Yaskawa INFORM job: ROBOT2.JBI

/JOB
//NAME ROBOT2
///FOLDERNAME INNE
//POS
///NPOS 25,25,0,0,0,0
///TOOL 0
///POSTYPE PULSE
///PULSE
C00000=-52530,-106772,-59840,25675,74247,58338
C00001=-30541,-61161,-38258,13058,102738,71922
C00002=-79491,-79946,-37138,33739,93735,85492
C00003=-123799,-144126,-48227,54109,53120,88750
C00004=-1049,-85507,-55311,-1240,88725,56676
C00005=10878,-82728,-51898,427,88114,60655
C00006=56233,-75375,-39159,-22430,94952,57482
C00007=77051,-120104,-53646,-32838,65753,47043
C00008=58715,-140663,-55283,-39550,38165,34197
C00009=-10070,-106255,-61443,11351,75991,18903
C00010=4969,-100505,-52101,12303,71167,23538
C00011=24839,-133484,-44655,5407,15605,27035
C00012=51428,-76992,-39319,-14366,84439,67888
C00013=5067,-115869,-54923,15370,51336,49727
C00014=2370,-61149,-31128,13691,95920,53857
C00015=14944,-75662,-39037,14855,81364,56560
C00016=52747,-124419,-44869,-21736,22441,76499
C00017=86721,-65113,-23109,-30643,87847,87051
C00018=67275,-41536,-10599,-20819,100364,86717
C00019=-49708,-95496,-27496,49930,72279,53724
C00020=-14954,-101056,-27545,59819,53704,58945
C00021=-14053,-108943,-20525,82453,42704,47577
C00022=3718,-38650,-2507,33351,95883,82801
C00023=23556,-89945,-42085,25883,63693,43192
C00024=75100,-38847,-12945,-13870,97090,65418
BC00000=140445,1007710,556393
BC00001=140445,1007710,556390
BC00002=140445,1007710,556390
BC00003=140445,1007710,556390
BC00004=140445,1007710,556390
BC00005=140445,1007709,556387
BC00006=140445,1007709,556387
BC00007=140445,1007709,556387
BC00008=140445,1007709,556387
BC00009=140445,1007709,556387
BC00010=140445,1007709,556385
BC00011=140445,1007709,556385
BC00012=140446,1007710,556382
BC00013=140446,1007710,556382
BC00014=140446,1007710,556382
BC00015=140446,1007710,556379
BC00016=140446,1007710,556379
BC00017=140446,1007710,556379
BC00018=140446,1007710,556379
BC00019=140446,1007710,556379
BC00020=140446,1007710,556376
BC00021=140446,1007710,556376
BC00022=140446,1007710,556376
BC00023=140446,1007710,556376
BC00024=140446,1007710,556376
//INST
///DATE 2023/10/04 15:13
///ATTR SC,RW
///GROUP1 RB1,BS1
NOP
*1
MOVJ C00000 BC00000 VJ=0.78 PL=0
MOVJ C00001 BC00001 VJ=0.78 PL=0
MOVJ C00002 BC00002 VJ=0.78 PL=0
MOVJ C00003 BC00003 VJ=0.78 PL=0
MOVJ C00004 BC00004 VJ=0.78 PL=0
*2
MOVJ C00005 BC00005 VJ=0.78 PL=0
MOVJ C00006 BC00006 VJ=0.78 PL=0
MOVJ C00007 BC00007 VJ=0.78 PL=0
MOVJ C00008 BC00008 VJ=0.78 PL=0
MOVJ C00009 BC00009 VJ=0.78 PL=0
*3
MOVJ C00010 BC00010 VJ=0.78 PL=0
MOVJ C00011 BC00011 VJ=0.78 PL=0
MOVJ C00012 BC00012 VJ=0.78 PL=0
MOVJ C00013 BC00013 VJ=0.78 PL=0
MOVJ C00014 BC00014 VJ=0.78 PL=0
*4
MOVJ C00015 BC00015 VJ=0.78 PL=0
MOVJ C00016 BC00016 VJ=0.78 PL=0
MOVJ C00017 BC00017 VJ=0.78 PL=0
MOVJ C00018 BC00018 VJ=0.78 PL=0
MOVJ C00019 BC00019 VJ=0.78 PL=0
*5
MOVJ C00020 BC00020 VJ=0.78 PL=0
MOVJ C00021 BC00021 VJ=0.78 PL=0
MOVJ C00022 BC00022 VJ=0.78 PL=0
MOVJ C00023 BC00023 VJ=0.78 PL=0
MOVJ C00024 BC00024 VJ=0.78 PL=0
END
